FUNCTION_BLOCK eigval_in (* Basic FB with empty ECC *)
  (* Standard: 61499-2 *)
  (* Version 1.0, 2020-08-19, Candra Wardaya, UGM *)
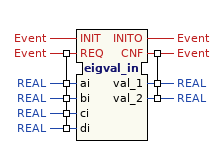
  EVENT_INPUT
    INIT;
    REQ WITH ai, bi, ci, di;
  END_EVENT
  EVENT_OUTPUT
    INITO;
    CNF WITH val_1, val_2;
  END_EVENT
  VAR_INPUT
    ai : REAL;
    bi : REAL;
    ci : REAL;
    di : REAL;
  END_VAR
  VAR_OUTPUT
    val_1 : REAL;
    val_2 : REAL;
  END_VAR
  VAR
    A : REAL; (* Internal Variable *)
    B : REAL; (* Internal Variable *)
    C : REAL; (* Internal Variable *)
    Di : REAL; (* Internal Variable *)
  END_VAR
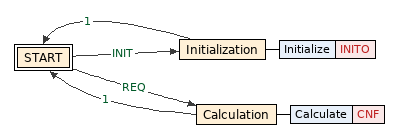
  EC_STATES
    START; (* Initial State *)
    Initialization : Initialize -> INITO;
    Calculation : Calculate -> CNF;
  END_STATES
  EC_TRANSITIONS
    START TO Initialization := INIT;
    Initialization TO START := 1;
    START TO Calculation := REQ;
    Calculation TO START := 1;
  END_TRANSITIONS
  ALGORITHM Initialize IN ST: (* New Algorithm *)

  END_ALGORITHM
  ALGORITHM Calculate IN ST: (* New Algorithm *)
A := 1;
B := -ai-di;
C := ai*di - bi*ci;

Di := EXPT(B,2) - 4*A*C;

val_2 := ((-B) + SQRT(Di))/(2*A);
val_1 := ((-B) - SQRT(Di))/(2*A);
  END_ALGORITHM
END_FUNCTION_BLOCK
